PROGRAM PRG_LI1K4_IP1
VAR
    {attribute 'pytmc' := '
        pv: LI1K4:IP1
        io: io
    '}
    fbLI1K4: FB_LIC;

    stSiBP: ST_BeamParams := PMPS_GVL.cstFullBeam;
    bInit: BOOL;
END_VAR


// Exclusion range specified by P. Walter 2021-5-19
//stSiBP.neVRange := F_eVExcludeRange(1.6E3, 3.2E3);
// Drop transmission to 20%
//stSiBP.nTran := 0.20;


//fbLI1K4.stOut.fPosition := 0.118;
fbLI1K4.stOut.bUseRawCounts := FALSE;
fbLI1K4.stOut.bValid := TRUE;
fbLI1K4.stOut.bMoveOk := TRUE;
fbLI1K4.stOut.stPMPS.sPmpsState := 'LI1K4:IP1-OUT';

//fbLI1K4.stMirror1.fPosition := -36.38;
fbLI1K4.stMirror1.bUseRawCounts := FALSE;
fbLI1K4.stMirror1.bValid := TRUE;
fbLI1K4.stMirror1.bMoveOk := TRUE;
fbLI1K4.stMirror1.stPMPS.sPmpsState := 'LI1K4:IP1-MIRROR1';

//fbLI1K4.stMirror2.fPosition := -70.38;
fbLI1K4.stMirror2.bUseRawCounts := FALSE;
fbLI1K4.stMirror2.bValid := TRUE;
fbLI1K4.stMirror2.bMoveOk := TRUE;
fbLI1K4.stMirror2.stPMPS.sPmpsState := 'LI1K4:IP1-MIRROR2';

//fbLI1K4.stTarget1.fPosition := -102.38;
fbLI1K4.stTarget1.bUseRawCounts := FALSE;
fbLI1K4.stTarget1.bValid := TRUE;
fbLI1K4.stTarget1.bMoveOk := TRUE;
fbLI1K4.stTarget1.stPMPS.sPmpsState := 'LI1K4:IP1-TARGET1';

IF NOT bInit THEN
   bInit := TRUE;
   fbLI1K4.stOut.fPosition := 0.118;
   fbLI1K4.stMirror1.fPosition := -36.38;
   fbLI1K4.stMirror2.fPosition := -70.38;
   fbLI1K4.stTarget1.fPosition := -102.38;
END_IF

fbLI1K4(
    fbArbiter := fbArbiter,
    fbFFHWO := fbFastFaultOutput1,
    stYStage := Main.M20,
    sDeviceName := 'LI1K4:IP1',
    sTransitionKey := 'LI1K4:IP1-TRANSITION',
    bEnableMotion := TRUE,
    bEnableBeamParams := TRUE,
    bEnablePositionLimits := TRUE,
);

END_PROGRAM

(* stored: Version 1.1.0.1, ProductVersion 3.1.4022.18
   POU PRG_LI1K4_IP1: Id {d1be7b36-4016-4b0e-aff6-a7c2bd7afb17}, SpecialFunc None *)
